(* IEC 61131-3 sources: AXOpen/src/components.pneumatics/app/SystemConstants, 2 files *)

(* ---- plc_line_IoAddresses.st ---- *)
CONFIGURATION IoAddresses
    VAR_GLOBAL

        // Module aes-d-bc-pnio/Slot_1
        aes_d_bc_pnio_Slot_1_Output AT %QB0 : aes_d_bc_pnio_Slot_1_Output_Layout;
    END_VAR
END_CONFIGURATION

TYPE
    aes_d_bc_pnio_Slot_1_Output_Layout : STRUCT
        Signals_0_0 AT %X0.0 : BOOL;
        Signals_0_1 AT %X0.1 : BOOL;
        Signals_0_2 AT %X0.2 : BOOL;
        Signals_0_3 AT %X0.3 : BOOL;
        Signals_0_4 AT %X0.4 : BOOL;
        Signals_0_5 AT %X0.5 : BOOL;
        Signals_0_6 AT %X0.6 : BOOL;
        Signals_0_7 AT %X0.7 : BOOL;
    END_STRUCT;
END_TYPE

(* ---- plc_line_HwIdentifiers.st ---- *)
CONFIGURATION HardwareIDs
    VAR_GLOBAL CONSTANT
        aes_d_bc_pnio_HwID : UINT := UINT#258;
        aes_d_bc_pnio_Rack_HwID : UINT := UINT#261;
        aes_d_bc_pnio_Slot_10_empty_slot_HwID : UINT := UINT#269;
        aes_d_bc_pnio_Slot_11_empty_slot_HwID : UINT := UINT#268;
        aes_d_bc_pnio_Slot_12_empty_slot_HwID : UINT := UINT#267;
        aes_d_bc_pnio_Slot_13_empty_slot_HwID : UINT := UINT#266;
        aes_d_bc_pnio_Slot_14_empty_slot_HwID : UINT := UINT#265;
        aes_d_bc_pnio_Slot_15_empty_slot_HwID : UINT := UINT#264;
        aes_d_bc_pnio_Slot_16_empty_slot_HwID : UINT := UINT#263;
        aes_d_bc_pnio_Slot_1_Valve_driver_4_valves_4_HwID : UINT := UINT#278;
        aes_d_bc_pnio_Slot_2_empty_slot_HwID : UINT := UINT#277;
        aes_d_bc_pnio_Slot_3_empty_slot_HwID : UINT := UINT#276;
        aes_d_bc_pnio_Slot_4_empty_slot_HwID : UINT := UINT#275;
        aes_d_bc_pnio_Slot_5_empty_slot_HwID : UINT := UINT#274;
        aes_d_bc_pnio_Slot_6_empty_slot_HwID : UINT := UINT#273;
        aes_d_bc_pnio_Slot_7_empty_slot_HwID : UINT := UINT#272;
        aes_d_bc_pnio_Slot_8_empty_slot_HwID : UINT := UINT#271;
        aes_d_bc_pnio_Slot_9_empty_slot_HwID : UINT := UINT#270;
        aes_d_bc_pnio_aes_d_bc_pnio_HwID : UINT := UINT#262;
        aes_d_bc_pnio_aes_d_bc_pnio_AES_Modul_HwID : UINT := UINT#279;
        aes_d_bc_pnio_aes_d_bc_pnio_PN_IO_HwID : UINT := UINT#257;
        aes_d_bc_pnio_aes_d_bc_pnio_PN_IO_Port_1_HwID : UINT := UINT#259;
        aes_d_bc_pnio_aes_d_bc_pnio_PN_IO_Port_2_HwID : UINT := UINT#260;
        plc_line_HwID : UINT := UINT#32;
        plc_line_Rail_0_HwID : UINT := UINT#280;
        plc_line_plc_line_HwID : UINT := UINT#48;
        plc_line_plc_line_CPU_display_1_HwID : UINT := UINT#54;
        plc_line_plc_line_Card_reader_writer_1_HwID : UINT := UINT#51;
        plc_line_plc_line_DP_interface_1_HwID : UINT := UINT#60;
        plc_line_plc_line_OPC_UA_1_HwID : UINT := UINT#117;
        plc_line_plc_line_PROFINET_interface_1_HwID : UINT := UINT#64;
        plc_line_plc_line_PROFINET_interface_1_Port_1_HwID : UINT := UINT#65;
        plc_line_plc_line_PROFINET_interface_1_Port_2_HwID : UINT := UINT#66;
        plc_line_plc_line_PROFINET_interface_2_HwID : UINT := UINT#72;
        plc_line_plc_line_PROFINET_interface_2_Port_3_HwID : UINT := UINT#73;
        plc_line_plc_line_Virtual_communication_interface_HwID : UINT := UINT#135;
        profinet_plc_line_HwID : UINT := UINT#256;

    END_VAR
END_CONFIGURATION
